DATA_BLOCK "DBVALVES"
{ S7_Optimized_Access := 'TRUE' }
VERSION : 0.1
NON_RETAIN
   VAR
      LAMP_TEST { S7_SetPoint := 'True'} : Bool;
      BR : Struct
         IMITATION { S7_SetPoint := 'False'} : "Tstate";   // [1] BR IMITATION
         FRAME_HOLDFAST { S7_SetPoint := 'False'} : "Tstate";   // [2] BR FRAME_HOLDFAST
         BUMPER { S7_SetPoint := 'False'} : "Tstate";   // [3] BR BUMPER
         CONTAINER_LATCH { S7_SetPoint := 'False'} : "Tstate";   // [4] BR CONTAINER_LATCH
         SWORD { S7_SetPoint := 'False'} : "Tstate";   // [5] BR SWORD
      END_STRUCT;
      ST1 : Struct
         STATION_RISING { S7_SetPoint := 'False'} : "Tstate";   // [6] ST1 STATION_RISING
         COVER_GUIDE { S7_SetPoint := 'False'} : "Tstate";   // [7] ST1 COVER_GUIDE
         COVER_LOCK { S7_SetPoint := 'False'} : "Tstate";   // [8] ST1 COVER_LOCK
         TAU_HOLDFAST_MOVEMENT { S7_SetPoint := 'False'} : "Tstate";   // [9] ST1 TAU_HOLDFAST_MOVEMENT
         TAU_HOLDFAST { S7_SetPoint := 'False'} : "Tstate";   // [10] ST1 TAU_HOLDFAST
         TAPE_RELEASE_MOVEMENT { S7_SetPoint := 'False'} : "Tstate";   // [11] ST1 TAPE_RELEASE_MOVEMENT
         TAPE_RELEASE { S7_SetPoint := 'False'} : "Tstate";   // [12] ST1 TAPE_RELEASE
         TAPE_OPEN { S7_SetPoint := 'False'} : "Tstate";   // [13] ST1 TAPE_OPEN
         CAMERA_MOVEMENT { S7_SetPoint := 'False'} : "Tstate";   // [14] ST1 CAMERA_MOVEMENT
         BASE_LOWERING { S7_SetPoint := 'False'} : "Tstate";   // [15] ST1 BASE_LOWERING
         TAPE_LOWERING { S7_SetPoint := 'False'} : "Tstate";   // [16] ST1 TAPE_LOWERING
         PINS_LOWERING { S7_SetPoint := 'False'} : "Tstate";   // [17] ST1 PINS_LOWERING
      END_STRUCT;
   END_VAR


BEGIN

END_DATA_BLOCK

